Staubli VAL3: create.pgx

public program create(num x_nDetNum (dimensions=1), string x_sTask (dimensions=1))
begin
  call init(x_nDetNum,x_sTask)
  taskCreate sTASK,100,detection()
end
